{attribute 'reflection'} 
FUNCTION_BLOCK FB_LAMP_DIMM IMPLEMENTS I_Lamp
VAR
	// Hardware control variables
	fOut : REAL;
	fInc : REAL:=0.5;
	iOutHw AT %Q*:INT;
	
	// Instance-path variable
    {attribute 'instance-path'} 
    {attribute 'noinit'} 
    sPath : STRING; 
END_VAR

METHOD OFF : BOOL
// Intensity in 0..100% variable fOut
fOut := fOut - fInc;
IF fOut < 0.0 THEN
	fOut := 0.0;
END_IF

// Conversion to hardware output 0..32767
iOutHw := LIMIT(0,REAL_TO_INT(fOut * 327.67), 32767);
END_METHOD

METHOD ON : BOOL
// Intensity in 0..100% variable fOut
fOut := fOut + fInc;
IF fOut > 100.0 THEN
	fOut := 100.0;
END_IF

// Conversion to hardware output 0..32767
iOutHw := LIMIT(0,REAL_TO_INT(fOut * 327.67), 32767);
END_METHOD

PROPERTY State : STRING
GET
State := CONCAT('Object: ', sPath);
State := CONCAT(State, ' State (%):');
State := CONCAT(State, REAL_TO_STRING(THIS^.fOut));
END_GET
END_PROPERTY

END_FUNCTION_BLOCK

(* stored: Version 1.1.0.1, ProductVersion 3.1.4024.6
   POU FB_LAMP_DIMM: Id {ef4dfccf-13f0-4f5d-beae-8fa75d59aa89}, SpecialFunc None
   Method OFF: Id {d33db4ea-238d-4d07-87b3-d7935e3aff2e}
   Method ON: Id {a36d9568-8c93-4146-8db2-1a2fa228ca51}
   Property State: Id {2e19e7c6-c212-489b-950d-b13dc8ea6993}
   Get Get: Id {b2b03c34-15f8-4434-8832-2387ec358a41} *)
